PROGRAM PRG_Eletric
VAR
END_VAR

END_PROGRAM

(* stored: Version 1.1.0.1, ProductVersion 3.1.4024.12
   POU PRG_Eletric: Id {bf5b672a-2b95-44a1-aca6-afef707f31cd}, SpecialFunc None *)
